// Implicitly generated code : DO NOT EDIT
FUNCTION CheckRangeSigned : DINT
VAR_INPUT
	value, lower, upper: DINT;
END_VAR

// Implicitly generated code : Only an Implementation suggestion
IF (value < lower) THEN
	CheckRangeSigned := lower;
	GVL_Checks.dCheckRangeSigned := GVL_Checks.dCheckRangeSigned + 1;
	ADSLOGSTR(4,'Checks critical error - DINT overflow.','');
ELSIF(value > upper) THEN
	CheckRangeSigned := upper;
	GVL_Checks.dCheckRangeSigned := GVL_Checks.dCheckRangeSigned + 1;
	ADSLOGSTR(4,'Checks critical error - DINT overflow.','');
ELSE
	CheckRangeSigned := value;
END_IF

END_FUNCTION

(* stored: Version 1.1.0.1, ProductVersion 3.1.4024.12
   POU CheckRangeSigned: Id {3f665f5c-f2d8-4cce-8287-4400ac7ad20d}, SpecialFunc CheckRangeSigned *)
